FUNCTION TryConvert_STRING_TO_STRING : BOOL
VAR_INPUT
	in : STRING;
	out : REFERENCE TO STRING;
END_VAR

out := in;
TryConvert_STRING_TO_STRING := TRUE;

END_FUNCTION

(* stored: Version 1.1.0.1, ProductVersion 3.1.4024.12
   POU TryConvert_STRING_TO_STRING: Id {cc1d70e8-7ccc-4b28-b188-0c92326cd832}, SpecialFunc None *)
